// TIA Portal V16 export
// export: Created 2024-06-17T18:37:12.687069Z, ExportSetting WithDefaults, DisplayName Totally Integrated Automation Portal, DisplayVersion V16, DisplayName TIA Portal Version Control Interface, DisplayVersion V16, DisplayName TIA Portal Openness, DisplayVersion V16, DisplayName STEP 7 Professional, DisplayVersion V16, DisplayName STEP 7 Safety, DisplayVersion V16, DisplayName WinCC Advanced, DisplayVersion V16
TYPE "Axis.Safety"
// stored: IsFailsafeCompliant true
   STRUCT
      Safety_Geral_Ok : Bool;   // Sistema de Segurança da Célula Restaurado
      BT_Emergência_01 : Bool;
      BT_Emergência_02 : Bool;
      BT_Emergência_03 : Bool;
      BT_Emergência_04 : Bool;
      BT_Emergência_05 : Bool;
      BT_Emergência_06 : Bool;
      BT_Emergência_07 : Bool;
      BT_Emergência_08 : Bool;
      BT_Emergência_09 : Bool;
      BT_Emergência_10 : Bool;
      Geral_BT_Emergência : Bool;   // Todos os Botões de Emergência Restaurados
      Corda_Emergência_01 : Bool;
      Corda_Emergência_02 : Bool;
      Corda_Emergência_03 : Bool;
      Corda_Emergência_04 : Bool;
      Corda_Emergência_05 : Bool;
      Corda_Emergência_06 : Bool;
      Corda_Emergência_07 : Bool;
      Corda_Emergência_08 : Bool;
      Corda_Emergência_09 : Bool;
      Corda_Emergência_10 : Bool;
      Geral_Corda_Emergência : Bool;   // Todos as Cordas de Emergência Restauradas
      Barreira_Luz_01 : Bool;
      Barreira_Luz_02 : Bool;
      Barreira_Luz_03 : Bool;
      Barreira_Luz_04 : Bool;
      Barreira_Luz_05 : Bool;
      Barreira_Luz_06 : Bool;
      Barreira_Luz_07 : Bool;
      Barreira_Luz_08 : Bool;
      Barreira_Luz_09 : Bool;
      Barreira_Luz_10 : Bool;
      Geral_Barreira_Luz : Bool;   // Todos as Barreiras de Luz Restauradas
      Portão_Segurança_01 : Bool;
      Portão_Segurança_02 : Bool;
      Portão_Segurança_03 : Bool;
      Portão_Segurança_04 : Bool;
      Portão_Segurança_05 : Bool;
      Portão_Segurança_06 : Bool;
      Portão_Segurança_07 : Bool;
      Portão_Segurança_08 : Bool;
      Portão_Segurança_09 : Bool;
      Portão_Segurança_10 : Bool;
      Geral_Portas_Segurança : Bool;   // Todos os Portas de Segurança Restauradas
   END_STRUCT;
END_TYPE
